PROGRAM MAIN
VAR
	bBool : BOOL := TRUE;
	
	eEventType1 : E_EventType := E_EventType.Alarm;
	eEventSeverity1 : TcEventSeverity := TcEventSeverity.Critical;
	nEventIdentity1 : UDINT := 0023654;
	sEventText1 : STRING(255) := '/!\ Scary event /!\';
	
	CsvPersistentEventStorage : FB_CsvPersistentEventStorage;
	EventLogger : EventLogger(CsvPersistentEventStorage);
END_VAR

(*
IF NOT bBool THEN
	UpdateEventTimestampWithSystemTime(stEvent := stFirstInstance);
	bBool := TRUE;
END_IF
*)

IF bBool THEN
	EventLogger.AddEvent(eEventType1, eEventSeverity1, nEventIdentity1, sEventText1);
	
	bBool := FALSE;
END_IF

CsvPersistentEventStorage();

END_PROGRAM

(* stored: Version 1.1.0.1, ProductVersion 3.1.4024.12
   POU MAIN: Id {05b5314c-6eef-4bab-81b0-22141dca3fa3}, SpecialFunc None *)
